Universal Robots PolyScope program: paletovani.urp

Program paletovani (installation=default directory=/home/ur/ursim/ursim-3.15.0.106151/programs createdIn=3.15.0.106151 lastSavedIn=3.15.0.106151 robotSerialNumber=2018359999)
Calibrated DH parameters: a=[0, -0.425, -0.39225, 0, 0, 0]; d=[0.089159, 0, 0, 0.10915, 0.09465, 0.0823]; alpha=[1.570796, 0, 0, 1.570796, -1.570796, 0]; deltaTheta=[0, 0, 0, 0, 0, 0]
Robot Program (runOnlyOnce=false)
  Pallet pattern(dimensionality=Square firstAxisCount=2 secondAxisCount=2 thirdAxisCount=5 motionType=MoveL speed=0.25 acceleration=1.2 useActiveTCP=true, counterVariable(name=cnt_1, initializeExpression=0), patternPoseVariable(name=pose_1), feature=Base, children(Waypoint(type=Fixed name=Corner1_1, position(joints=-1.5879243055926722, -1.9841497580157679, -2.282199207936422, -0.47143870988954717, 1.5954264402389526, -0.018224541340963185 pose=-0.11451424317374755, -0.43056219778754795, 0.03983958932140483, -0.0012211811904130855, 3.1162765300146344, 0.03889226399566927), poseInFeatureCoordinates=[-0.114514, -0.430562, 0.03984, -0.001221, 3.116277, 0.038892], outputFlangePose=[-0.114514, -0.430562, 0.03984, -0.001221, 3.116277, 0.038892]), Waypoint(type=Fixed name=Corner2_1, position(joints=-1.414156738911764, -1.9669764677630823, -2.3193722406970423, -0.4467981497394007, 1.5994465351104736, 0.15555839240550995 pose=-0.0401159096047915, -0.43056226172127293, 0.039839664971381125, -0.0012212780118130966, 3.1162764588224094, 0.03889215777556428), poseInFeatureCoordinates=[-0.040116, -0.430562, 0.03984, -0.001221, 3.116276, 0.038892], outputFlangePose=[-0.040116, -0.430562, 0.03984, -0.001221, 3.116276, 0.038892]), Waypoint(type=Fixed name=Corner3_1, position(joints=-1.372298542653219, -1.8474138418780726, -2.5592833201037806, -0.3252323309527796, 1.6002899408340454, 0.1974259316921234 pose=-0.04011598479265722, -0.34176391961497427, 0.039839718265610294, -0.00122105447489096, 3.116276498844161, 0.03889184482622922), poseInFeatureCoordinates=[-0.040116, -0.341764, 0.03984, -0.001221, 3.116276, 0.038892], outputFlangePose=[-0.040116, -0.341764, 0.03984, -0.001221, 3.116276, 0.038892]), Waypoint(type=Fixed name=Corner4_1, position(joints=-1.6221807638751429, -1.8723304907428187, -2.504814688359396, -0.3614705244647425, 1.5945422649383545, -0.052479092274801076 pose=-0.12491438789698896, -0.3417639617724935, 0.039839775144130646, -0.0012203866837396302, 3.1162765006526114, 0.0388914370911562), poseInFeatureCoordinates=[-0.124914, -0.341764, 0.03984, -0.00122, 3.116277, 0.038891], outputFlangePose=[-0.124914, -0.341764, 0.03984, -0.00122, 3.116277, 0.038891]))); actionSequence(name=PalletSequence motionType=MoveL speed=0.25 acceleration=1.2 useActiveTCP=true, anchorWaypoint(type=Fixed name=PatternPoint_1, position(joints=-1.4581268469439905, -1.9900081793414515, -2.3658908049212855, -0.3784874121295374, 1.5985064506530762, 0.1115812361240387 pose=-0.06091607400929564, -0.41216220281173666, 0.025439597082378224, -0.0012207025758573912, 3.1162765142669553, 0.03889248202811647), poseInFeatureCoordinates=[-0.060916, -0.412162, 0.02544, -0.001221, 3.116277, 0.038892], outputFlangePose=[-0.060916, -0.412162, 0.02544, -0.001221, 3.116277, 0.038892]), feature=Base, children(Waypoint(type=Fixed name=Approach_1, position(joints=-1.6135662237750452, -1.7500823179828089, -2.275019947682516, -0.7133081595050257, 1.5947673320770264, -0.043865505849019826 pose=-0.1249143687565776, -0.41216218601971505, 0.11943804327910608, -0.001221107454260285, 3.1162764355860793, 0.03889176868407514), poseInFeatureCoordinates=[-0.124914, -0.412162, 0.119438, -0.001221, 3.116276, 0.038892], outputFlangePose=[-0.124914, -0.412162, 0.119438, -0.001221, 3.116276, 0.038892]), Waypoint=PatternPoint_1, Contributed(strategyProgramNodeType=Gripper strategyURCapDeveloper=URCaps R us Inc. strategyURCapName=Sps, dataModel(steps=66, test=false, width=20)), Wait(type=Sleep, waitTime=0.01), Waypoint(type=Fixed name=Exit_1, position(joints=-1.4581268469439905, -1.4535415808307093, -2.0989392439471644, -1.1819050947772425, 1.5985064506530762, 0.1115812361240387 pose=-0.06091606837300858, -0.41216225307141785, 0.27023644904722444, -0.001220712854459426, 3.1162764700594994, 0.0388917430743868), poseInFeatureCoordinates=[-0.060916, -0.412162, 0.270236, -0.001221, 3.116276, 0.038892], outputFlangePose=[-0.060916, -0.412162, 0.270236, -0.001221, 3.116276, 0.038892])))
    Pattern -> pattern
    AnchoredSequence -> PalletSequence
  Pallet pattern(dimensionality=Square firstAxisCount=2 secondAxisCount=2 thirdAxisCount=5 motionType=MoveL speed=0.25 acceleration=1.2 useActiveTCP=true, counterVariable(name=cnt_2, initializeExpression=0), patternPoseVariable(name=pose_2), feature=Base, children(Waypoint(type=Fixed name=Corner1_2, position(joints=2.272653341293335, -2.0260260740863245, -1.8220503965960901, -0.9461029211627405, 1.597933292388916, 3.719329357147217 pose=-0.2881975694601801, 0.506472608761095, 0.12651524115587995, -0.19127801613841833, 3.1060400350091437, -0.12736000477883272), poseInFeatureCoordinates=[-0.288198, 0.506473, 0.126515, -0.191278, 3.10604, -0.12736], outputFlangePose=[-0.288198, 0.506473, 0.126515, -0.191278, 3.10604, -0.12736]), Waypoint(type=Fixed name=Corner2_2, position(joints=2.191936731338501, -2.1577704588519495, -1.5997193495379847, -1.0386059919940394, 1.59125816822052, 3.6388661861419678 pose=-0.28680849646217765, 0.5854379197898563, 0.1265150579677916, -0.1912781396500836, 3.1060397151030563, -0.12736077098345788), poseInFeatureCoordinates=[-0.286808, 0.585438, 0.126515, -0.191278, 3.10604, -0.127361], outputFlangePose=[-0.286808, 0.585438, 0.126515, -0.191278, 3.10604, -0.127361]), Waypoint(type=Fixed name=Corner3_2, position(joints=2.283984661102295, -2.2371886412249964, -1.460383717213766, -1.0962956587420862, 1.5988572835922241, 3.7306272983551025 pose=-0.36639458132706015, 0.5868378329000508, 0.12651502606792914, -0.19127790560317032, 3.1060397632409638, -0.12736046961333822), poseInFeatureCoordinates=[-0.366395, 0.586838, 0.126515, -0.191278, 3.10604, -0.12736], outputFlangePose=[-0.366395, 0.586838, 0.126515, -0.191278, 3.10604, -0.12736]), Waypoint(type=Fixed name=Corner4_2, position(joints=2.4587080478668213, -2.0053990522967737, -1.8574445883380335, -0.9249232451068323, 1.6125813722610474, 3.904918670654297 pose=-0.36903969223015337, 0.4364627629417905, 0.12651510838910757, -0.1912780681977865, 3.106039808911038, -0.12736052881951088), poseInFeatureCoordinates=[-0.36904, 0.436463, 0.126515, -0.191278, 3.10604, -0.127361], outputFlangePose=[-0.36904, 0.436463, 0.126515, -0.191278, 3.10604, -0.127361]))); actionSequence(name=PalletSequence motionType=MoveL speed=0.25 acceleration=1.2 useActiveTCP=true, anchorWaypoint(type=Fixed name=PatternPoint_2, position(joints=2.393716812133789, -2.024557892476217, -1.9910414854632776, -0.7747162024127405, 1.6076027154922485, 3.8400681018829346 pose=-0.3134493683213822, 0.4355174014243806, 0.08096893846251758, -0.19127830396762333, 3.106039678227615, -0.1273605748049413), poseInFeatureCoordinates=[-0.313449, 0.435517, 0.080969, -0.191278, 3.10604, -0.127361], outputFlangePose=[-0.313449, 0.435517, 0.080969, -0.191278, 3.10604, -0.127361]), feature=Base, children(Waypoint(type=Fixed name=Approach_2, position(joints=2.4587080478668213, -1.8248360792743128, -1.6796162764178675, -1.2833145300494593, 1.6125813722610474, 3.904918670654297 pose=-0.3690396311448185, 0.4364627132908319, 0.27216740481118956, -0.19127806819779117, 3.106039808911038, -0.12736052881951718), poseInFeatureCoordinates=[-0.36904, 0.436463, 0.272167, -0.191278, 3.10604, -0.127361], outputFlangePose=[-0.36904, 0.436463, 0.272167, -0.191278, 3.10604, -0.127361]), Waypoint=PatternPoint_2, Contributed(strategyProgramNodeType=Gripper strategyURCapDeveloper=URCaps R us Inc. strategyURCapName=Sps, dataModel(steps=66, test=false, width=30)), Wait(type=Sleep, waitTime=0.01), Waypoint(type=Fixed name=Exit_2, position(joints=2.393716812133789, -1.6790626684771937, -1.435355011616842, -1.6758979002581995, 1.6076027154922485, 3.8400681018829346 pose=-0.3134493967083909, 0.4355174278556851, 0.43296570344847796, -0.19127830396762122, 3.106039678227615, -0.1273605748049415), poseInFeatureCoordinates=[-0.313449, 0.435517, 0.432966, -0.191278, 3.10604, -0.127361], outputFlangePose=[-0.313449, 0.435517, 0.432966, -0.191278, 3.10604, -0.127361])))
    Pattern -> pattern
    AnchoredSequence -> PalletSequence
  MoveJ speed 60 deg/s, acceleration 80 deg/s^2 (useActiveTCP=true)
    Waypoint Waypoint_1: TCP in base x=-411.308 y=-155.054 z=434.224 mm, rx=0.6027 ry=-2.2893 rz=-0.4385 rad; joints [-138.489, -77.488, -112.093, -47.246, 54.885, -88.754] deg
  Pallet pattern(dimensionality=Square firstAxisCount=2 secondAxisCount=2 thirdAxisCount=5 motionType=MoveL speed=0.25 acceleration=1.2 useActiveTCP=true, counterVariable(name=cnt_3, initializeExpression=0), patternPoseVariable(name=pose_3), feature=Base, children(Waypoint(type=Fixed name=Corner1_2, position(joints=2.272653341293335, -2.0260260740863245, -1.8220503965960901, -0.9461029211627405, 1.597933292388916, 3.719329357147217 pose=-0.2881975694601801, 0.506472608761095, 0.12651524115587995, -0.19127801613841833, 3.1060400350091437, -0.12736000477883272), poseInFeatureCoordinates=[-0.288198, 0.506473, 0.126515, -0.191278, 3.10604, -0.12736], outputFlangePose=[-0.288198, 0.506473, 0.126515, -0.191278, 3.10604, -0.12736]), Waypoint(type=Fixed name=Corner2_2, position(joints=2.191936731338501, -2.1577704588519495, -1.5997193495379847, -1.0386059919940394, 1.59125816822052, 3.6388661861419678 pose=-0.28680849646217765, 0.5854379197898563, 0.1265150579677916, -0.1912781396500836, 3.1060397151030563, -0.12736077098345788), poseInFeatureCoordinates=[-0.286808, 0.585438, 0.126515, -0.191278, 3.10604, -0.127361], outputFlangePose=[-0.286808, 0.585438, 0.126515, -0.191278, 3.10604, -0.127361]), Waypoint(type=Fixed name=Corner3_2, position(joints=2.283984661102295, -2.2371886412249964, -1.460383717213766, -1.0962956587420862, 1.5988572835922241, 3.7306272983551025 pose=-0.36639458132706015, 0.5868378329000508, 0.12651502606792914, -0.19127790560317032, 3.1060397632409638, -0.12736046961333822), poseInFeatureCoordinates=[-0.366395, 0.586838, 0.126515, -0.191278, 3.10604, -0.12736], outputFlangePose=[-0.366395, 0.586838, 0.126515, -0.191278, 3.10604, -0.12736]), Waypoint(type=Fixed name=Corner4_2, position(joints=2.4587080478668213, -2.0053990522967737, -1.8574445883380335, -0.9249232451068323, 1.6125813722610474, 3.904918670654297 pose=-0.36903969223015337, 0.4364627629417905, 0.12651510838910757, -0.1912780681977865, 3.106039808911038, -0.12736052881951088), poseInFeatureCoordinates=[-0.36904, 0.436463, 0.126515, -0.191278, 3.10604, -0.127361], outputFlangePose=[-0.36904, 0.436463, 0.126515, -0.191278, 3.10604, -0.127361]))); actionSequence(name=PalletSequence motionType=MoveL speed=0.25 acceleration=1.2 useActiveTCP=true, anchorWaypoint(type=Fixed name=PatternPoint_2, position(joints=2.393716812133789, -2.024557892476217, -1.9910414854632776, -0.7747162024127405, 1.6076027154922485, 3.8400681018829346 pose=-0.3134493683213822, 0.4355174014243806, 0.08096893846251758, -0.19127830396762333, 3.106039678227615, -0.1273605748049413), poseInFeatureCoordinates=[-0.313449, 0.435517, 0.080969, -0.191278, 3.10604, -0.127361], outputFlangePose=[-0.313449, 0.435517, 0.080969, -0.191278, 3.10604, -0.127361]), feature=Base, children(Waypoint(type=Fixed name=Approach_2, position(joints=2.4587080478668213, -1.8248360792743128, -1.6796162764178675, -1.2833145300494593, 1.6125813722610474, 3.904918670654297 pose=-0.3690396311448185, 0.4364627132908319, 0.27216740481118956, -0.19127806819779117, 3.106039808911038, -0.12736052881951718), poseInFeatureCoordinates=[-0.36904, 0.436463, 0.272167, -0.191278, 3.10604, -0.127361], outputFlangePose=[-0.36904, 0.436463, 0.272167, -0.191278, 3.10604, -0.127361]), Waypoint=PatternPoint_2, Contributed(strategyProgramNodeType=Gripper strategyURCapDeveloper=URCaps R us Inc. strategyURCapName=Sps, dataModel(steps=66, test=false, width=20)), Wait(type=Sleep, waitTime=0.01), Waypoint(type=Fixed name=Exit_2, position(joints=2.393716812133789, -1.6790626684771937, -1.435355011616842, -1.6758979002581995, 1.6076027154922485, 3.8400681018829346 pose=-0.3134493967083909, 0.4355174278556851, 0.43296570344847796, -0.19127830396762122, 3.106039678227615, -0.1273605748049415), poseInFeatureCoordinates=[-0.313449, 0.435517, 0.432966, -0.191278, 3.10604, -0.127361], outputFlangePose=[-0.313449, 0.435517, 0.432966, -0.191278, 3.10604, -0.127361])))
    Pattern -> pattern
    AnchoredSequence -> PalletSequence
  Pallet pattern(dimensionality=Square firstAxisCount=2 secondAxisCount=2 thirdAxisCount=5 motionType=MoveL speed=0.25 acceleration=1.2 useActiveTCP=true, counterVariable(name=cnt_4, initializeExpression=0), patternPoseVariable(name=pose_4), feature=Base, children(Waypoint(type=Fixed name=Corner1_1, position(joints=-1.5879243055926722, -1.9841497580157679, -2.282199207936422, -0.47143870988954717, 1.5954264402389526, -0.018224541340963185 pose=-0.11451424317374755, -0.43056219778754795, 0.03983958932140483, -0.0012211811904130855, 3.1162765300146344, 0.03889226399566927), poseInFeatureCoordinates=[-0.114514, -0.430562, 0.03984, -0.001221, 3.116277, 0.038892], outputFlangePose=[-0.114514, -0.430562, 0.03984, -0.001221, 3.116277, 0.038892]), Waypoint(type=Fixed name=Corner2_1, position(joints=-1.414156738911764, -1.9669764677630823, -2.3193722406970423, -0.4467981497394007, 1.5994465351104736, 0.15555839240550995 pose=-0.0401159096047915, -0.43056226172127293, 0.039839664971381125, -0.0012212780118130966, 3.1162764588224094, 0.03889215777556428), poseInFeatureCoordinates=[-0.040116, -0.430562, 0.03984, -0.001221, 3.116276, 0.038892], outputFlangePose=[-0.040116, -0.430562, 0.03984, -0.001221, 3.116276, 0.038892]), Waypoint(type=Fixed name=Corner3_1, position(joints=-1.372298542653219, -1.8474138418780726, -2.5592833201037806, -0.3252323309527796, 1.6002899408340454, 0.1974259316921234 pose=-0.04011598479265722, -0.34176391961497427, 0.039839718265610294, -0.00122105447489096, 3.116276498844161, 0.03889184482622922), poseInFeatureCoordinates=[-0.040116, -0.341764, 0.03984, -0.001221, 3.116276, 0.038892], outputFlangePose=[-0.040116, -0.341764, 0.03984, -0.001221, 3.116276, 0.038892]), Waypoint(type=Fixed name=Corner4_1, position(joints=-1.6221807638751429, -1.8723304907428187, -2.504814688359396, -0.3614705244647425, 1.5945422649383545, -0.052479092274801076 pose=-0.12491438789698896, -0.3417639617724935, 0.039839775144130646, -0.0012203866837396302, 3.1162765006526114, 0.0388914370911562), poseInFeatureCoordinates=[-0.124914, -0.341764, 0.03984, -0.00122, 3.116277, 0.038891], outputFlangePose=[-0.124914, -0.341764, 0.03984, -0.00122, 3.116277, 0.038891]))); actionSequence(name=PalletSequence motionType=MoveL speed=0.25 acceleration=1.2 useActiveTCP=true, anchorWaypoint(type=Fixed name=PatternPoint_1, position(joints=-1.4581268469439905, -1.9900081793414515, -2.3658908049212855, -0.3784874121295374, 1.5985064506530762, 0.1115812361240387 pose=-0.06091607400929564, -0.41216220281173666, 0.025439597082378224, -0.0012207025758573912, 3.1162765142669553, 0.03889248202811647), poseInFeatureCoordinates=[-0.060916, -0.412162, 0.02544, -0.001221, 3.116277, 0.038892], outputFlangePose=[-0.060916, -0.412162, 0.02544, -0.001221, 3.116277, 0.038892]), feature=Base, children(Waypoint(type=Fixed name=Approach_1, position(joints=-1.6135662237750452, -1.7500823179828089, -2.275019947682516, -0.7133081595050257, 1.5947673320770264, -0.043865505849019826 pose=-0.1249143687565776, -0.41216218601971505, 0.11943804327910608, -0.001221107454260285, 3.1162764355860793, 0.03889176868407514), poseInFeatureCoordinates=[-0.124914, -0.412162, 0.119438, -0.001221, 3.116276, 0.038892], outputFlangePose=[-0.124914, -0.412162, 0.119438, -0.001221, 3.116276, 0.038892]), Waypoint=PatternPoint_1, Contributed(strategyProgramNodeType=Gripper strategyURCapDeveloper=URCaps R us Inc. strategyURCapName=Sps, dataModel(steps=66, test=false, width=30)), Wait(type=Sleep, waitTime=0.01), Waypoint(type=Fixed name=Exit_1, position(joints=-1.4581268469439905, -1.4535415808307093, -2.0989392439471644, -1.1819050947772425, 1.5985064506530762, 0.1115812361240387 pose=-0.06091606837300858, -0.41216225307141785, 0.27023644904722444, -0.001220712854459426, 3.1162764700594994, 0.0388917430743868), poseInFeatureCoordinates=[-0.060916, -0.412162, 0.270236, -0.001221, 3.116276, 0.038892], outputFlangePose=[-0.060916, -0.412162, 0.270236, -0.001221, 3.116276, 0.038892])))
    Pattern -> pattern
    AnchoredSequence -> PalletSequence
